# B&R Automation Studio project MappAssetInt (part 2)

#### exAssetIntCore.st
```iecst
// -------------------------------------------------------------------------------------------
// Core function block
FUNCTION_BLOCK exAssetIntCore
	// -------------------------------------------------------------------------------------------
	// Reset everything when enable is false
	IF NOT Enable THEN
		Active := FALSE;
		exLink.IsCoreActive := FALSE;
		StatusID := ERR_FUB_ENABLE_FALSE;
		Internal.State := exASSETINT_STATE_INIT_1;
		CreateLoggerEntry(exASSETINT_LOG_INFO, ADR('function block disabled'), Logger);
		RETURN;
	END_IF

	CASE Internal.State OF

		// -------------------------------------------------------------------------------------------
		// Wait for enable
		// -------------------------------------------------------------------------------------------
		exASSETINT_STATE_INIT_1:
			IF Enable THEN
				CreateLoggerEntry(exASSETINT_LOG_INFO, ADR('function block enabled'), Logger);

				// Make sure we have remanent buffer
				IF ADR(exLink) = 0 THEN
					// Set status, remember state, go to error state
					StatusID := CreateErrorState(ERR_ASSET_LINK, ADR('ERR: exLink is 0'), Logger, exCOM_SEV_ERROR,  ADR(Internal.State), ADR(Info.Diag.StatusID));
					RETURN;
				END_IF
				// Make sure we have a configuration
				IF ADR(Configuration) = 0 THEN
					// Set status, remember state, go to error state
					StatusID := CreateErrorState(ERR_ASSET_LINK, ADR('ERR: No configuation attached'), Logger, exCOM_SEV_ERROR,  ADR(Internal.State), ADR(Info.Diag.StatusID));
					RETURN;
				END_IF

				// -------------------------------------------------------------------------------------------
				// Transfer start values
				exLink.RecordCount := 0;
				exLink.JobStatistics.JobName := Parameters.Job;
				exLink.JobStatistics.CurrentUser := Parameters.CurrentUser;
				exLink.JobStatistics.AdditionalData := Parameters.AdditionalData;
				Internal.JobPieceCounterOld := PieceCounter;
				Internal.JobRejectCounterOld := RejectCounter;

				exLink.ShiftStatistics.CurrentUser := Parameters.CurrentUser;
				exLink.ShiftStatistics.AdditionalData := Parameters.AdditionalData;
				Internal.ShiftPieceCounterOld := PieceCounter;
				Internal.ShiftRejectCounterOld := RejectCounter;

				// -------------------------------------------------------------------------------------------
				// Reset error, status and function and internal blocks
				Error := FALSE;
				StatusID := ERR_OK;
				Internal.CreateDirStructure(Enable := FALSE);
				Internal.CreateMemory(Enable := FALSE);
				Internal.ReadEventData(Enable := FALSE);
				Internal.WriteEventData(Enable := FALSE);
				Internal.ReadEventData(Enable := FALSE);
				Internal.WriteEventData(Enable := FALSE);

				// -------------------------------------------------------------------------------------------
				// Check shift configuration for errors
				IF NOT exAssetIntCheckShiftData(Configuration, Logger, ADR(Internal.State), ADR(StatusID), ADR(Info.Diag.StatusID)) THEN
					RETURN;
				END_IF

				// -------------------------------------------------------------------------------------------
				// Create folder structure and read event data only after boot
				IF Internal.InitAfterBoot THEN
					Internal.State := exASSETINT_STATE_INIT_4;
				ELSE
					Internal.State := exASSETINT_STATE_INIT_2;
				END_IF
			END_IF

			// -------------------------------------------------------------------------------------------
			// Create folder structure
			// -------------------------------------------------------------------------------------------
		exASSETINT_STATE_INIT_2:
			Internal.CreateDirStructure.Enable := TRUE;
			Internal.CreateDirStructure.Device := DeviceName;
			Internal.CreateDirStructure.Logger := Logger;
			Internal.CreateDirStructure();

			// -------------------------------------------------------------------------------------------
			// Folder structure successful created
			IF Internal.CreateDirStructure.Status = ERR_OK THEN
				CreateLoggerEntry(exASSETINT_LOG_INFO, ADR('create folder structure ok'), Logger);
				Internal.State := exASSETINT_STATE_INIT_3;

				// Error
			ELSIF Internal.CreateDirStructure.Status <> ERR_FUB_BUSY THEN
				// Set status, remember state, go to error state
				StatusID := CreateErrorState(Internal.CreateDirStructure.Status, ADR('ERR: create folder structure'), Logger, exCOM_SEV_ERROR,  ADR(Internal.State), ADR(Info.Diag.StatusID));
			END_IF

			// -------------------------------------------------------------------------------------------
			// Create internal memory
			// -------------------------------------------------------------------------------------------
		exASSETINT_STATE_INIT_3:
			Internal.CreateMemory.Enable := TRUE;
			Internal.CreateMemory.Size := CORE_EVENT_NUM_MAX*SIZEOF(Internal.RecordData);
			Internal.CreateMemory.Logger := Logger;
			Internal.CreateMemory();

			// -------------------------------------------------------------------------------------------
			// Memory structure successful created
			IF Internal.CreateMemory.Status = ERR_OK THEN
				CreateLoggerEntry(exASSETINT_LOG_INFO, ADR('create internal memory ok'), Logger);
				exLink.MemoryDb := Internal.CreateMemory.MemoryDb;
				exLink.MemoryJob := Internal.CreateMemory.MemoryJob;
				exLink.MemoryShift := Internal.CreateMemory.MemoryShift;
				exLink.MemoryTimeline := Internal.CreateMemory.MemoryTimeline;
				Internal.InitAfterBoot := TRUE;
				Internal.State := exASSETINT_STATE_INIT_4;

				// Error
			ELSIF Internal.CreateMemory.Status <> ERR_FUB_BUSY THEN
				// Set status, remember state, go to error state
				StatusID := CreateErrorState(Internal.CreateMemory.Status, ADR('ERR: create internal memory'), Logger, exCOM_SEV_ERROR,  ADR(Internal.State), ADR(Info.Diag.StatusID));
			END_IF

			// -------------------------------------------------------------------------------------------
			// Read event data
			// -------------------------------------------------------------------------------------------
		exASSETINT_STATE_INIT_4:
			Internal.ReadEventData.Enable := TRUE;
			Internal.ReadEventData.Device := DeviceName;
			Internal.ReadEventData.Memory := exLink.MemoryDb;
			Internal.ReadEventData.Logger := Logger;
			Internal.ReadEventData();

			// Read events successful
			IF Internal.ReadEventData.Status = ERR_OK THEN
				CreateLoggerEntry(exASSETINT_LOG_INFO, ADR('read stored events ok'), Logger);

				// -------------------------------------------------------------------------------------------
				// Get record count, calculate next entry
				exLink.RecordCount := Internal.ReadEventData.RecordCount;
				IF exLink.RecordCount > 0 THEN
					// Get last entry, make correction if necessary
					brsmemcpy(ADR(Internal.RecordData), exLink.MemoryDb + (exLink.RecordCount - 1)*SIZEOF(Internal.RecordData), SIZEOF(Internal.RecordData));
					brsstrcpy(ADR(Internal.TmpStr1), ADR(Internal.RecordData.FileName) + FindInstr(ADR(Internal.RecordData.FileName), ADR('#')) + 1);
					Internal.RecordNext := DINT_TO_UINT(brsatoi(ADR(Internal.TmpStr1))) + 1;
					IF Internal.RecordNext >= CORE_EVENT_NUM_MAX THEN
						Internal.RecordNext := 0;
					END_IF
				END_IF

				// -------------------------------------------------------------------------------------------
				// Remember start called time
				Internal.TimeLastCallShift := clock_ms();
				Internal.TimeLastCallProduction := clock_ms();

				// -------------------------------------------------------------------------------------------
				// Refresh UI data, finish up
				exLink.RefreshJobUI := TRUE;
				exLink.RefreshShiftUI := TRUE;
				exLink.RefreshTimelineUI := TRUE;
				Internal.State := exASSETINT_STATE_IDLE;

				// Error
			ELSIF Internal.ReadEventData.Status <> ERR_FUB_BUSY THEN
				// Set status, remember state, go to error state
				StatusID := CreateErrorState(Internal.ReadEventData.Status, ADR('ERR: read stored events'), Logger, exCOM_SEV_ERROR,  ADR(Internal.State), ADR(Info.Diag.StatusID));
			END_IF

			// -------------------------------------------------------------------------------------------
			// Wait for new event
			// -------------------------------------------------------------------------------------------
		exASSETINT_STATE_IDLE:
			// Set core active, reset read write function blocks
			Active := TRUE;
			exLink.IsCoreActive := TRUE;
			Internal.ReadEventData(Enable := FALSE);
			Internal.WriteEventData(Enable := FALSE);

			// Update time information
			Internal.DTGetTime_0(enable := TRUE);
			DT_TO_DTStructure(Internal.DTGetTime_0.DT1, ADR(Internal.DT_TO_DTStructure_0));
			Internal.TimeOfDay := UDINT_TO_TOD((USINT_TO_UDINT(Internal.DT_TO_DTStructure_0.hour) * 3600000) + (USINT_TO_UDINT(Internal.DT_TO_DTStructure_0.minute) * 60000) + (USINT_TO_UDINT(Internal.DT_TO_DTStructure_0.second) * 1000));

			// Set stats timer
			Internal.StatsRefresh.IN := TRUE;
			Internal.StatsRefresh.PT := Configuration.CalculationTimeBase/10;
			Internal.StatsRefresh();

			// -------------------------------------------------------------------------------------------
			// Track current shift
			Internal.ShiftName := '';
			Internal.ShiftId := -1;
			FOR Internal.x := 0 TO SIZEOF(Configuration.Shifts)/SIZEOF(Configuration.Shifts[0]) - 1 DO
				// Shift ends on same day
				IF Configuration.Shifts[Internal.x].TotalTime.Start < Configuration.Shifts[Internal.x].TotalTime.End THEN
					IF Internal.TimeOfDay >= Configuration.Shifts[Internal.x].TotalTime.Start AND Internal.TimeOfDay <= Configuration.Shifts[Internal.x].TotalTime.End THEN
						Internal.ShiftName := Configuration.Shifts[Internal.x].Name;
						Internal.ShiftId := UINT_TO_SINT(Internal.x);
						EXIT;
					END_IF
					// Shift ends next day
				ELSE
					IF Internal.TimeOfDay >= Configuration.Shifts[Internal.x].TotalTime.Start OR Internal.TimeOfDay <= Configuration.Shifts[Internal.x].TotalTime.End THEN
						Internal.ShiftName := Configuration.Shifts[Internal.x].Name;
						Internal.ShiftId := UINT_TO_SINT(Internal.x);
						EXIT;
					END_IF
				END_IF
			END_FOR;

			// -------------------------------------------------------------------------------------------
			// Track current shift scheduled downtime
			IF exLink.ShiftId >= 0 THEN
				FOR Internal.x := 0 TO SIZEOF(Configuration.Shifts[exLink.ShiftId].ScheduledDowntime)/SIZEOF(Configuration.Shifts[exLink.ShiftId].ScheduledDowntime[0]) - 1 DO
					// Make sure we have a valid configuration
					IF TOD_TO_UDINT(Configuration.Shifts[exLink.ShiftId].ScheduledDowntime[Internal.x].Start) <> 0 OR TOD_TO_UDINT(Configuration.Shifts[exLink.ShiftId].ScheduledDowntime[Internal.x].End) <> 0 THEN
						// Downtime ends on same day
						IF Configuration.Shifts[exLink.ShiftId].ScheduledDowntime[Internal.x].Start < Configuration.Shifts[exLink.ShiftId].ScheduledDowntime[Internal.x].End THEN
							IF Internal.TimeOfDay >= Configuration.Shifts[exLink.ShiftId].ScheduledDowntime[Internal.x].Start AND Internal.TimeOfDay < Configuration.Shifts[exLink.ShiftId].ScheduledDowntime[Internal.x].End THEN
								Downtime := exASSETINT_SCHEDULED_DOWNTIME;
								DowntimeReason := Configuration.Shifts[exLink.ShiftId].ScheduledDowntime[Internal.x].Reason;
								EXIT;
							END_IF
						ELSE
							IF Internal.TimeOfDay >= Configuration.Shifts[exLink.ShiftId].ScheduledDowntime[Internal.x].Start OR Internal.TimeOfDay < Configuration.Shifts[exLink.ShiftId].ScheduledDowntime[Internal.x].End THEN
								Downtime := exASSETINT_SCHEDULED_DOWNTIME;
								DowntimeReason := Configuration.Shifts[exLink.ShiftId].ScheduledDowntime[Internal.x].Reason;
								EXIT;
							END_IF
						END_IF
					END_IF
				END_FOR;
			END_IF

			// -------------------------------------------------------------------------------------------
			// Handle shift change
			IF exLink.ShiftStatistics.ShiftName <> Internal.ShiftName THEN
				// Transfer stats to record, make sure structures are allignent
				brsmemset(ADR(Internal.RecordData), 0, SIZEOF(Internal.RecordData));

				IF Internal.ShiftName <> '' THEN
					Internal.TmpStr1 := 'new shift started ';
					brsstrcat(ADR(Internal.TmpStr1), ADR(Internal.ShiftName));
					CreateLoggerEntry(exASSETINT_LOG_INFO, ADR(Internal.TmpStr1), Logger);
				ELSIF exLink.ShiftStatistics.ShiftName <> '' THEN
					Internal.TmpStr1 := 'shift ended ';
					brsstrcat(ADR(Internal.TmpStr1), ADR(exLink.ShiftStatistics.ShiftName));
					CreateLoggerEntry(exASSETINT_LOG_INFO, ADR(Internal.TmpStr1), Logger);
				END_IF

				// Only store data when shift name was not empty
				IF exLink.ShiftStatistics.ShiftName <> '' THEN
					// Collect data for record
					Internal.RecordData.EventType := RecordTypeShift;
					Internal.RecordData.TimeStart := exLink.ShiftStatistics.StartTime;
					Internal.DT_TO_DTStructure_0.hour := UDINT_TO_USINT(TOD_TO_UDINT(Configuration.Shifts[exLink.ShiftId].TotalTime.End)/3600000);
					Internal.DT_TO_DTStructure_0.minute := UDINT_TO_USINT((TOD_TO_UDINT(Configuration.Shifts[exLink.ShiftId].TotalTime.End) - Internal.DT_TO_DTStructure_0.hour*3600000)/60000);
					Internal.RecordData.TimeEnd := DTStructure_TO_DT(ADR(Internal.DT_TO_DTStructure_0));
					Internal.RecordData.CurrentUser := exLink.ShiftStatistics.CurrentUser;
					Internal.RecordData.AdditionalData := exLink.ShiftStatistics.AdditionalData;
					Internal.RecordData.ShiftName := exLink.ShiftStatistics.ShiftName;
					Internal.RecordData.JobName := exLink.JobStatistics.JobName;
					Internal.RecordData.TotalPieces := exLink.ShiftStatistics.TotalPieces;
					Internal.RecordData.GoodPieces := exLink.ShiftStatistics.GoodPieces;
					Internal.RecordData.RejectPieces := exLink.ShiftStatistics.RejectPieces;
					Internal.RecordData.BadPieceRate := exLink.ShiftStatistics.BadPieceRate;
					Internal.RecordData.TargetPieces := exLink.ShiftStatistics.TargetPieces;
					Internal.RecordData.TotalTime := exLink.ShiftStatistics.TotalTime;
					Internal.RecordData.ScheduledDowntime := exLink.ShiftStatistics.ScheduledDowntime;
					Internal.RecordData.UnscheduledDowntime := exLink.ShiftStatistics.UnscheduledDowntime;
					Internal.RecordData.Uptime := exLink.ShiftStatistics.Uptime;
					Internal.RecordData.GoodProductionTime := exLink.ShiftStatistics.GoodProductionTime;
					Internal.RecordData.NominalProductionTime := exLink.ShiftStatistics.NominalProductionTime;
					Internal.RecordData.NominalProductionTimeRate := exLink.ShiftStatistics.NominalProductionTimeRate;
					Internal.RecordData.UnscheduledDowntimeRate := exLink.ShiftStatistics.UnscheduledDowntimeRate;
					Internal.RecordData.CurrentProductionRate := exLink.ShiftStatistics.CurrentProductionRate;

					Internal.State := exASSETINT_STATE_STORE_EVENT;
				END_IF

				// Remember job start time
				IF exLink.JobStatistics.StartTime = DT#1970-01-01-00:00:00 THEN
					exLink.JobStatistics.StartTime := Internal.DTGetTime_0.DT1;
				END_IF

				// Reset stats
				brsmemset(ADR(Info.ShiftStatistics), 0, SIZEOF(Info.ShiftStatistics));
				brsmemset(ADR(exLink.ShiftStatistics), 0, SIZEOF(exLink.ShiftStatistics));

				exLink.ShiftTotalTime := 0;
				exLink.ShiftDowntimeScheduled := 0;
				exLink.ShiftDowntimeUnscheduled := 0;

				// Transfer data to shift stats
				exLink.ShiftId := Internal.ShiftId;
				exLink.ShiftStatistics.StartTime := Internal.DTGetTime_0.DT1;
				exLink.ShiftStatistics.ShiftName := Internal.ShiftName;
				exLink.ShiftStatistics.CurrentUser := Parameters.CurrentUser;
				exLink.ShiftStatistics.AdditionalData := Parameters.AdditionalData;
			END_IF

			// -------------------------------------------------------------------------------------------
			// Calculate shift and job statistics
			IF Internal.ShiftName <> '' THEN

				// Calculate new stats
				IF Internal.StatsRefresh.Q THEN
					// Get time difference between calls
					Internal.DiffLastCallShift := DiffT(clock_ms(), Internal.TimeLastCallShift);
					Internal.TimeLastCallShift := clock_ms();

					// Handle diff timer overflow
					IF Internal.DiffLastCallShift = 16#FFFFFFFF THEN
						CreateLoggerEntry(exASSETINT_LOG_INFO, ADR('diff timer overflow'), Logger);
					ELSE

						// Do not count when downtime is active
						IF Downtime = exASSETINT_NO_DOWNTIME THEN
							// Transfer job counter data
							IF Internal.JobPieceCounterOld <= PieceCounter THEN
								exLink.JobStatistics.TotalPieces := exLink.JobStatistics.TotalPieces + (PieceCounter - Internal.JobPieceCounterOld);
							ELSE
								CreateLoggerEntry(exASSETINT_LOG_ERROR, ADR('job piece count overflow'), Logger);
								exLink.JobStatistics.TotalPieces := exLink.JobStatistics.TotalPieces + (16#FFFFFFFF - Internal.JobPieceCounterOld + PieceCounter);
							END_IF

							IF Internal.JobRejectCounterOld <= RejectCounter THEN
								exLink.JobStatistics.RejectPieces := exLink.JobStatistics.RejectPieces + (RejectCounter - Internal.JobRejectCounterOld);
							ELSE
								CreateLoggerEntry(exASSETINT_LOG_ERROR, ADR('job reject count overflow'), Logger);
								exLink.JobStatistics.RejectPieces := exLink.JobStatistics.RejectPieces + (16#FFFFFFFF - Internal.JobRejectCounterOld + RejectCounter);
							END_IF
						END_IF
						Internal.JobPieceCounterOld := PieceCounter;
						Internal.JobRejectCounterOld := RejectCounter;
						CalcStatsJob(exLink, Internal.DiffLastCallShift, Downtime, Parameters, ADR(Info.JobStatistics));

						// Do not count when downtime is active
						IF Downtime = exASSETINT_NO_DOWNTIME THEN
							// Transfer shift counter data
							IF Internal.ShiftPieceCounterOld <= PieceCounter THEN
								exLink.ShiftStatistics.TotalPieces := exLink.ShiftStatistics.TotalPieces + (PieceCounter - Internal.ShiftPieceCounterOld);
							ELSE
								CreateLoggerEntry(exASSETINT_LOG_ERROR, ADR('shift piece count overflow'), Logger);
								exLink.ShiftStatistics.TotalPieces := exLink.ShiftStatistics.TotalPieces + (16#FFFFFFFF - Internal.ShiftPieceCounterOld + PieceCounter);
							END_IF

							IF Internal.ShiftRejectCounterOld <= RejectCounter THEN
								exLink.ShiftStatistics.RejectPieces := exLink.ShiftStatistics.RejectPieces + (RejectCounter - Internal.ShiftRejectCounterOld);
							ELSE
								CreateLoggerEntry(exASSETINT_LOG_ERROR, ADR('shift reject count overflow'), Logger);
								exLink.ShiftStatistics.RejectPieces := exLink.ShiftStatistics.RejectPieces + (16#FFFFFFFF - Internal.ShiftRejectCounterOld + RejectCounter);
							END_IF
						END_IF
						Internal.ShiftPieceCounterOld := PieceCounter;
						Internal.ShiftRejectCounterOld := RejectCounter;
						CalcStatsShift(exLink, Internal.DiffLastCallShift, Downtime, Parameters, ADR(Info.ShiftStatistics));

						// Transfer shift data to main function block
						CurrentProductionRate := exLink.ShiftStatistics.CurrentProductionRate;
						NominalProductionTimeRate := exLink.ShiftStatistics.NominalProductionTimeRate;
						BadPieceRate := exLink.ShiftStatistics.BadPieceRate;
						ScheduledDowntimeRate := exLink.ShiftStatistics.ScheduledDowntimeRate;
						UnscheduledDowntimeRate := exLink.ShiftStatistics.UnscheduledDowntimeRate;

					END_IF
				END_IF

				// When no shift is active
			ELSE
				// Dont count when no shift is active, reset last call
				Internal.ShiftPieceCounterOld := PieceCounter;
				Internal.ShiftRejectCounterOld := RejectCounter;
				Internal.JobPieceCounterOld := PieceCounter;
				Internal.JobRejectCounterOld := RejectCounter;

				Internal.TimeLastCallShift := clock_ms();
			END_IF

			// -------------------------------------------------------------------------------------------
			// Handle production state change
			IF Internal.State <> exASSETINT_STATE_STORE_EVENT THEN
				IF (exLink.ShiftStatistics.ShiftName <> exLink.ProductionShiftName) OR (exLink.JobStatistics.JobName <> exLink.ProductionJobName AND exLink.ShiftId >= 0) OR (Downtime <> exLink.ProductionDowntime AND exLink.ShiftId >= 0) THEN
					// Create log message
					Internal.TmpStr1 := 'production state changed from ';
					IF exLink.ProductionState = exASSETINT_STATE_NO_SHIFT_ACTIVE THEN
						brsstrcat(ADR(Internal.TmpStr1), ADR('no shift to '));
					ELSIF exLink.ProductionState = exASSETINT_STATE_UPTIME THEN
						brsstrcat(ADR(Internal.TmpStr1), ADR('uptime to '));
					ELSIF exLink.ProductionState = exASSETINT_STATE_SCHDL_DOWNTIME THEN
						brsstrcat(ADR(Internal.TmpStr1), ADR('scheduled dt to '));
					ELSE
						brsstrcat(ADR(Internal.TmpStr1), ADR('unscheduled dt to '));
					END_IF

					// Transfer stats to record, make sure structures are allignent
					brsmemset(ADR(Internal.RecordData), 0, SIZEOF(Internal.RecordData));

					// Collect data for record
					Internal.RecordData.TimeStart := exLink.ProductionStateStart;
					Internal.RecordData.TimeEnd := Internal.DTGetTime_0.DT1;
					Internal.RecordData.ShiftName := exLink.ProductionShiftName;
					Internal.RecordData.JobName := exLink.ProductionJobName;
					Internal.RecordData.EventType := UDINT_TO_UINT(exLink.ProductionState + 2);

					Internal.ProductionTotalTime := LREAL_TO_UDINT(exLink.ProductionTotalTime/1000);
					Internal.RecordData.TotalTime.Hours := Internal.ProductionTotalTime/3600;
					Internal.RecordData.TotalTime.Minutes := UDINT_TO_USINT((Internal.ProductionTotalTime - Internal.RecordData.TotalTime.Hours*3600)/60);
					Internal.RecordData.TotalTime.Seconds := UDINT_TO_USINT(Internal.ProductionTotalTime - Internal.RecordData.TotalTime.Hours*3600 - Internal.RecordData.TotalTime.Minutes*60);

					// State change is new job
					IF (exLink.JobStatistics.JobName <> exLink.ProductionJobName) THEN
						brsstrcat(ADR(Internal.TmpStr1), ADR('new job > '));
						brsstrcat(ADR(Internal.TmpStr1), ADR(exLink.JobStatistics.JobName));
						exLink.ProductionState := exASSETINT_STATE_UPTIME;

						// State change is to no shift
					ELSIF (exLink.ProductionShiftName <> '' AND exLink.ShiftStatistics.ShiftName = '') THEN
						brsstrcat(ADR(Internal.TmpStr1), ADR('no shift'));
						exLink.ProductionState := exASSETINT_STATE_NO_SHIFT_ACTIVE;

						// State change is to uptime
					ELSIF (exLink.ProductionShiftName = '' AND exLink.ShiftStatistics.ShiftName <> '') THEN
						brsstrcat(ADR(Internal.TmpStr1), ADR('uptime'));
						exLink.ProductionState := exASSETINT_STATE_UPTIME;

						// State is shift change
					ELSIF (exLink.ProductionShiftName <> exLink.ShiftStatistics.ShiftName) THEN
						brsstrcat(ADR(Internal.TmpStr1), ADR('new shift'));
						exLink.ProductionState := exASSETINT_STATE_UPTIME;

						// State change is downtime
					ELSE
						IF Downtime = exASSETINT_NO_DOWNTIME THEN
							brsstrcat(ADR(Internal.TmpStr1), ADR('no downtime'));
						ELSIF Downtime = exASSETINT_SCHEDULED_DOWNTIME THEN
							brsstrcat(ADR(Internal.TmpStr1), ADR('scheduled dt > '));
							brsstrcat(ADR(Internal.TmpStr1), ADR(DowntimeReason));
						ELSE
							brsstrcat(ADR(Internal.TmpStr1), ADR('unscheduled dt > '));
							brsstrcat(ADR(Internal.TmpStr1), ADR(DowntimeReason));
						END_IF

						IF exLink.ProductionState = exASSETINT_STATE_SCHDL_DOWNTIME OR exLink.ProductionState = exASSETINT_STATE_UNSCH_DOWNTIME THEN
							Internal.RecordData.AdditionalData := DowntimeReason;
						END_IF
						exLink.ProductionState := UDINT_TO_UINT(Downtime + 1);
					END_IF
					CreateLoggerEntry(exASSETINT_LOG_INFO, ADR(Internal.TmpStr1), Logger);

					exLink.ProductionShiftName :=exLink.ShiftStatistics.ShiftName;
					exLink.ProductionJobName := exLink.JobStatistics.JobName;
					exLink.ProductionDowntime := Downtime;

					// Skip after cold start
					IF exLink.ProductionStateStart <> DT#1970-01-01-00:00:00 THEN
						exLink.ProductionStateStart := Internal.DTGetTime_0.DT1;
						exLink.ProductionTotalTime := 0;

						// Create new event
						Internal.State := exASSETINT_STATE_STORE_EVENT;

						// Just remember start time after cold start
					ELSE
						exLink.ProductionStateStart := Internal.DTGetTime_0.DT1;
					END_IF

				END_IF
			END_IF
			// Remember production duration
			IF Internal.StatsRefresh.Q THEN
				// Get time difference between calls
				Internal.DiffLastCallProduction := DiffT(clock_ms(), Internal.TimeLastCallProduction);
				Internal.TimeLastCallProduction := clock_ms();
				IF Internal.DiffLastCallProduction = 16#FFFFFFFF THEN
					CreateLoggerEntry(exASSETINT_LOG_INFO, ADR('diff timer overflow'), Logger);
				ELSE
					exLink.ProductionTotalTime := exLink.ProductionTotalTime + Internal.DiffLastCallProduction;
				END_IF
			END_IF

			// -------------------------------------------------------------------------------------------
			// Handle update command
			IF EDGEPOS(Update) THEN
				CreateLoggerEntry(exASSETINT_LOG_INFO, ADR('update command triggered'), Logger);

				// -------------------------------------------------------------------------------------------
				// Check shift configuration for errors
				IF NOT exAssetIntCheckShiftData(Configuration, Logger, ADR(Internal.State), ADR(StatusID), ADR(Info.Diag.StatusID)) THEN
					RETURN;
				END_IF

				// Job has changed
				IF Parameters.Job <> exLink.JobStatistics.JobName THEN
					Internal.TmpStr1 := 'new job started ';
					brsstrcat(ADR(Internal.TmpStr1), ADR(Parameters.Job));
					CreateLoggerEntry(exASSETINT_LOG_INFO, ADR(Internal.TmpStr1), Logger);

					CommandBusy := TRUE;
					CommandDone := FALSE;
					UpdateDone := FALSE;

					// Transfer stats to record, make sure structures are allignent
					brsmemset(ADR(Internal.RecordData), 0, SIZEOF(Internal.RecordData));

					// Collect data for record
					Internal.RecordData.EventType := RecordTypeJob;
					Internal.RecordData.TimeStart := exLink.JobStatistics.StartTime;
					Internal.RecordData.TimeEnd := Internal.DTGetTime_0.DT1;
					Internal.RecordData.CurrentUser := exLink.JobStatistics.CurrentUser;
					Internal.RecordData.AdditionalData := exLink.JobStatistics.AdditionalData;
					Internal.RecordData.ShiftName := exLink.ShiftStatistics.ShiftName;
					Internal.RecordData.JobName := exLink.JobStatistics.JobName;
					Internal.RecordData.TotalPieces := exLink.JobStatistics.TotalPieces;
					Internal.RecordData.GoodPieces := exLink.JobStatistics.GoodPieces;
					Internal.RecordData.RejectPieces := exLink.JobStatistics.RejectPieces;
					Internal.RecordData.BadPieceRate := exLink.JobStatistics.BadPieceRate;
					Internal.RecordData.TotalTime := exLink.JobStatistics.TotalTime;
					Internal.RecordData.ScheduledDowntime := exLink.JobStatistics.ScheduledDowntime;
					Internal.RecordData.UnscheduledDowntime := exLink.JobStatistics.UnscheduledDowntime;
					Internal.RecordData.Uptime := exLink.JobStatistics.Uptime;
					Internal.RecordData.GoodProductionTime := exLink.JobStatistics.GoodProductionTime;
					Internal.RecordData.NominalProductionTime := exLink.JobStatistics.NominalProductionTime;
					Internal.RecordData.NominalProductionTimeRate := exLink.JobStatistics.NominalProductionTimeRate;
					Internal.RecordData.UnscheduledDowntimeRate := exLink.JobStatistics.UnscheduledDowntimeRate;
					Internal.RecordData.CurrentProductionRate := exLink.JobStatistics.CurrentProductionRate;

					// Reset stats and remember new start time
					brsmemset(ADR(Info.JobStatistics), 0, SIZEOF(Info.JobStatistics));
					brsmemset(ADR(exLink.JobStatistics), 0, SIZEOF(exLink.JobStatistics));

					exLink.JobTotalTime := 0;
					exLink.JobDowntimeScheduled := 0;
					exLink.JobDowntimeUnscheduled := 0;

					// Transfer data to job stats
					exLink.JobStatistics.StartTime := Internal.DTGetTime_0.DT1;
					exLink.JobStatistics.JobName := Parameters.Job;
					exLink.JobStatistics.CurrentUser := Parameters.CurrentUser;
					exLink.JobStatistics.AdditionalData := Parameters.AdditionalData;

					Internal.State := exASSETINT_STATE_STORE_EVENT;
				ELSE
					CommandBusy := FALSE;
					CommandDone := TRUE;
					UpdateDone := TRUE;
				END_IF
			END_IF

			IF NOT Update THEN
				UpdateDone := FALSE;
			END_IF

			// -------------------------------------------------------------------------------------------
			// Handle reset command
			IF EDGEPOS(Reset) THEN
				CreateLoggerEntry(exASSETINT_LOG_INFO, ADR('reset command triggered'), Logger);

				CommandBusy := TRUE;
				CommandDone := FALSE;

				// Reset stats
				brsmemset(ADR(Info.JobStatistics), 0, SIZEOF(Info.JobStatistics));
				brsmemset(ADR(exLink.JobStatistics), 0, SIZEOF(exLink.JobStatistics));

				exLink.JobTotalTime := 0;
				exLink.JobDowntimeScheduled := 0;
				exLink.JobDowntimeUnscheduled := 0;

				// Transfer data to job stats
				exLink.JobStatistics.StartTime := Internal.DTGetTime_0.DT1;
				exLink.JobStatistics.JobName := Parameters.Job;
				exLink.JobStatistics.CurrentUser := Parameters.CurrentUser;
				exLink.JobStatistics.AdditionalData := Parameters.AdditionalData;

				// Reset stats
				brsmemset(ADR(Info.ShiftStatistics), 0, SIZEOF(Info.ShiftStatistics));
				brsmemset(ADR(exLink.ShiftStatistics), 0, SIZEOF(exLink.ShiftStatistics));

				exLink.ShiftTotalTime := 0;
				exLink.ShiftDowntimeScheduled := 0;
				exLink.ShiftDowntimeUnscheduled := 0;

				// Transfer data to shift stats
				exLink.ShiftId := Internal.ShiftId;
				exLink.ShiftStatistics.StartTime := Internal.DTGetTime_0.DT1;
				exLink.ShiftStatistics.ShiftName := Internal.ShiftName;
				exLink.ShiftStatistics.CurrentUser := Parameters.CurrentUser;
				exLink.ShiftStatistics.AdditionalData := Parameters.AdditionalData;

				CommandBusy := FALSE;
				CommandDone := TRUE;
			END_IF

			// -------------------------------------------------------------------------------------------
			// Handle export command
			IF EDGEPOS(Export) THEN

				CommandBusy := TRUE;
				CommandDone := FALSE;
				ExportDone := FALSE;

				Internal.State := exASSETINT_STATE_EXPORT_EVENTS;
			END_IF

			IF NOT Export THEN
				ExportDone := FALSE;
			END_IF

			// -------------------------------------------------------------------------------------------
			// Reset refresh timer
			IF Internal.StatsRefresh.Q THEN
				// Set stats timer
				Internal.StatsRefresh.IN := FALSE;
				Internal.StatsRefresh();
			END_IF

			IF Update = FALSE AND Export = FALSE AND Reset = FALSE THEN
				CommandDone := FALSE;
			END_IF

			// -------------------------------------------------------------------------------------------
			// Store new event
			// -------------------------------------------------------------------------------------------
		exASSETINT_STATE_STORE_EVENT:
			Internal.WriteEventData.Enable := TRUE;
			Internal.WriteEventData.Device := StorageName;
			Internal.WriteEventData.Logger := Logger;
			Internal.WriteEventData.RecordData := ADR(Internal.RecordData);
			Internal.WriteEventData.RecordNext := Internal.RecordNext;
			Internal.WriteEventData();

			// -------------------------------------------------------------------------------------------
			// Event successful created
			IF Internal.WriteEventData.Status = ERR_OK THEN
				CreateLoggerEntry(exASSETINT_LOG_INFO, ADR('create new event ok'), Logger);

				// Calculate new last record and record count
				Internal.RecordNext := Internal.RecordNext + 1;
				IF Internal.RecordNext >= CORE_EVENT_NUM_MAX THEN
					Internal.RecordNext := 0;
				END_IF
				// Copy new record into memeory
				IF exLink.RecordCount < CORE_EVENT_NUM_MAX THEN
					exLink.RecordCount := exLink.RecordCount + 1;
				ELSE
					brsmemmove(exLink.MemoryDb, exLink.MemoryDb + SIZEOF(Internal.RecordData), SIZEOF(Internal.RecordData)*(exLink.RecordCount - 1));
				END_IF
				brsmemcpy(exLink.MemoryDb + SIZEOF(Internal.RecordData)*(exLink.RecordCount - 1), ADR(Internal.RecordData), SIZEOF(Internal.RecordData));

				// Refrehs UI data, finish up
				exLink.RefreshJobUI := TRUE;
				exLink.RefreshShiftUI := TRUE;
				exLink.RefreshTimelineUI := TRUE;

				UpdateDone := TRUE;
				CommandBusy := FALSE;
				CommandDone := TRUE;

				StatusID := ERR_OK;
				Internal.State := exASSETINT_STATE_IDLE;

				// Error
			ELSIF Internal.WriteEventData.Status <> ERR_FUB_BUSY THEN
				// Set status, remember state, go to error state
				StatusID := CreateErrorState(Internal.WriteEventData.Status, ADR('ERR: create new event'), Logger, exCOM_SEV_ERROR,  ADR(Internal.State), ADR(Info.Diag.StatusID));
			END_IF

			// -------------------------------------------------------------------------------------------
			// Export all events
			// -------------------------------------------------------------------------------------------
		exASSETINT_STATE_EXPORT_EVENTS:
			Internal.ExportEventData.Enable := TRUE;
			Internal.ExportEventData.Device := DeviceName;
			Internal.ExportEventData.Logger := Logger;
			Internal.ExportEventData.RecordCount := exLink.RecordCount;
			Internal.ExportEventData.Memory := exLink.MemoryDb;
			Internal.ExportEventData.Configuration := Configuration.Export;
			Internal.ExportEventData();

			// -------------------------------------------------------------------------------------------
			// Event successful created
			IF Internal.ExportEventData.Status = ERR_OK THEN
				CreateLoggerEntry(exASSETINT_LOG_INFO, ADR('export events ok'), Logger);

				ExportDone := TRUE;
				CommandBusy := FALSE;
				CommandDone := TRUE;

				StatusID := ERR_OK;
				Internal.State := exASSETINT_STATE_IDLE;

				// Error
			ELSIF Internal.ExportEventData.Status <> ERR_FUB_BUSY THEN
				// Set status, remember state, go to error state
				StatusID := CreateErrorState(Internal.ExportEventData.Status, ADR('ERR: export events'), Logger, exCOM_SEV_ERROR,  ADR(Internal.State), ADR(Info.Diag.StatusID));
			END_IF

			// -------------------------------------------------------------------------------------------
			// Error state
			// -------------------------------------------------------------------------------------------
		exASSETINT_STATE_ERROR:

			// Reset error state
			IF EDGEPOS(ErrorReset) THEN
				Internal.StateError := exASSETINT_STATE_NONE;
				Internal.State := exASSETINT_STATE_INIT_1;
			END_IF
	END_CASE;

END_FUNCTION_BLOCK
```

#### exAssetIntCoreConfig.st
```iecst
// -------------------------------------------------------------------------------------------
// File version 1004
// -------------------------------------------------------------------------------------------
// Config function block
FUNCTION_BLOCK exAssetIntCoreConfig
	// -------------------------------------------------------------------------------------------
	// Reset everything when enable is false
	IF NOT Enable THEN
		Active := FALSE;
		StatusID := ERR_FUB_ENABLE_FALSE;
		Internal.State := exASSETINT_STATE_INIT_1;
		CreateLoggerEntry(exASSETINT_LOG_INFO, ADR('function block disabled'), Logger);
		RETURN;
	END_IF

	// -------------------------------------------------------------------------------------------
	// Permanent watch critical values
	IF Internal.State <> exASSETINT_STATE_ERROR THEN
		// Make sure we have a configuration
		IF ADR(Configuration) = 0 THEN
			// Set status, remember state, go to error state
			StatusID := CreateErrorState(ERR_ASSET_LINK, ADR('ERR: No configuation attached'), Logger, exCOM_SEV_ERROR, ADR(Internal.State), ADR(Info.Diag.StatusID));
			RETURN;
		END_IF
		// Make sure we have a device name
		IF ADR(DeviceName) = 0 THEN
			// Set status, remember state, go to error state
			StatusID := CreateErrorState(ERR_ASSET_LINK, ADR('ERR: No device name attached'), Logger, exCOM_SEV_ERROR, ADR(Internal.State), ADR(Info.Diag.StatusID));
			RETURN;
		END_IF
	END_IF

	CASE Internal.State OF

		// -------------------------------------------------------------------------------------------
		// Wait for enable
		exASSETINT_STATE_INIT_1:
			IF Enable THEN
				CreateLoggerEntry(exASSETINT_LOG_INFO, ADR('function block enabled'), Logger);

				// Reset error and status
				brsmemset(ADR(Info.Diag), 0, SIZEOF(Info.Diag));
				Error := FALSE;
				StatusID := ERR_OK;
				CommandBusy := FALSE;
				CommandDone := FALSE;

				Internal.State := exASSETINT_STATE_IDLE;
			END_IF

			// -------------------------------------------------------------------------------------------
			// Wait for new event
		exASSETINT_STATE_IDLE:
			Active := TRUE;

			// Handle configuration load command
			IF EDGEPOS(Load) THEN
				CreateLoggerEntry(exASSETINT_LOG_INFO, ADR('command load configuration'), Logger);
				CommandBusy := TRUE;
				CommandDone := FALSE;

				Internal.State := exASSETINT_STATE_LOAD_CFG;
			END_IF

			// Handle configuration save command
			IF EDGEPOS(Save) THEN
				CreateLoggerEntry(exASSETINT_LOG_INFO, ADR('command save configuration'), Logger);
				CommandBusy := TRUE;
				CommandDone := FALSE;

				Internal.State := exASSETINT_STATE_SAVE_CFG;
			END_IF

			IF Load = FALSE AND Save = FALSE THEN
				CommandDone := FALSE;
			END_IF

		// -------------------------------------------------------------------------------------------
		// Load configuration
		exASSETINT_STATE_LOAD_CFG:
			Internal.ReadConfiguration.Enable := TRUE;
			Internal.ReadConfiguration.Device := ADR(DeviceName);
			Internal.ReadConfiguration.Logger := Logger;
			Internal.ReadConfiguration();

			// Event successful created
			IF Internal.ReadConfiguration.Status = ERR_OK THEN
				CreateLoggerEntry(exASSETINT_LOG_INFO, ADR('load configuration ok'), Logger);
				Configuration := Internal.ReadConfiguration.Configuration;

				CommandBusy := FALSE;
				CommandDone := TRUE;
				StatusID := ERR_OK;

				Internal.State := exASSETINT_STATE_IDLE;

			// Error
			ELSIF Internal.ReadConfiguration.Status <> ERR_FUB_BUSY THEN
				// Set status, remember state, go to error state
				StatusID := CreateErrorState(Internal.ReadConfiguration.Status, ADR('ERR: load configuration'), Logger, exCOM_SEV_ERROR,  ADR(Internal.State), ADR(Info.Diag.StatusID));
			END_IF

			// -------------------------------------------------------------------------------------------
			// Save configuration
		exASSETINT_STATE_SAVE_CFG:
			Internal.WriteConfiguration.Enable := TRUE;
			Internal.WriteConfiguration.Device := ADR(DeviceName);
			Internal.WriteConfiguration.Logger := Logger;
			Internal.WriteConfiguration.Configuration := Configuration;
			Internal.WriteConfiguration();

			// Event successful created
			IF Internal.WriteConfiguration.Status = ERR_OK THEN
				CreateLoggerEntry(exASSETINT_LOG_INFO, ADR('save configuration ok'), Logger);

				CommandBusy := FALSE;
				CommandDone := TRUE;
				StatusID := ERR_OK;

				Internal.State := exASSETINT_STATE_IDLE;

			// Error
			ELSIF Internal.WriteConfiguration.Status <> ERR_FUB_BUSY THEN
				// Set status, remember state, go to error state
				StatusID := CreateErrorState(Internal.WriteConfiguration.Status, ADR('ERR: save configuration'), Logger, exCOM_SEV_ERROR,  ADR(Internal.State), ADR(Info.Diag.StatusID));
			END_IF

		// -------------------------------------------------------------------------------------------
		// Error state
		exASSETINT_STATE_ERROR:
			Internal.WriteConfiguration.Enable := FALSE;
			Internal.WriteConfiguration();
			Internal.ReadConfiguration.Enable := FALSE;
			Internal.ReadConfiguration();

			IF EDGEPOS(ErrorReset) THEN
				Internal.StateError := exASSETINT_STATE_NONE;
				Internal.State := exASSETINT_STATE_INIT_1;
			END_IF
	END_CASE;
END_FUNCTION_BLOCK
```

#### exAssetIntUI.st
```iecst
// -------------------------------------------------------------------------------------------
// Job UI function block
FUNCTION_BLOCK exAssetIntJobListUI
	// -------------------------------------------------------------------------------------------
	// Reset everything when enable is false
	IF NOT Enable THEN
		StatusID := ERR_FUB_ENABLE_FALSE;
		Active := FALSE;
		Internal.State := exASSETINT_STATE_INIT_1;
		CreateLoggerEntry(exASSETINT_LOG_INFO, ADR('function block disabled'), Logger);
		RETURN;
	END_IF

	CASE Internal.State OF

		// -------------------------------------------------------------------------------------------
		// Wait for enable
		exASSETINT_STATE_INIT_1:
			IF Enable THEN
				CreateLoggerEntry(exASSETINT_LOG_INFO, ADR('function block enabled'), Logger);

				// Check prerequisites, exLink and buffers
				IF NOT exAssetIntCheckPreq(exLink, Logger, ADR(Internal.State), ADR(StatusID), ADR(Info.Diag.StatusID)) THEN
					RETURN;
				END_IF

				// Reset error and status
				Error := FALSE;
				StatusID := ERR_OK;
				Internal.SortingStartTimeOld := UDINT_TO_DINT(16#FFFFFFFF);

				// Reset filter settings
				exAssetIntFilterReset(ADR(UIConnect.Filter));

				Internal.State := exASSETINT_STATE_IDLE;
			END_IF

			// -------------------------------------------------------------------------------------------
			// Wait for new event
		exASSETINT_STATE_IDLE:
			// Set status
			UIConnect.Status := exASSETINT_UI_STATUS_IDLE;
			Active := TRUE;

			// Handle dialog window
			Internal.State := exAssetIntFilterListUI(ADR(UIConnect.Filter), ADR(UIConnect.Status), Logger);

			// Handle sorting direction change
			IF UISetup.SortingStartTime <> Internal.SortingStartTimeOld AND exLink.RecordCount > 0 THEN
				Internal.State := exASSETINT_STATE_UI_BUFFER;
			END_IF
			Internal.SortingStartTimeOld := UISetup.SortingStartTime;

			// Handle page up and down
			exAssetIntScrollListUI(Internal.RecordCount, UI_JOB_LIST_IDX, ADR(UIConnect.Output.PageUp), ADR(UIConnect.Output.PageDown), ADR(UIConnect.Output.StepUp), ADR(UIConnect.Output.StepDown), ADR(Internal.RecordStart), ADR(Internal.State));

			// Wait for core task to call update command
			IF exLink.RefreshJobUI AND exLink.RecordCount > 0 THEN
				Internal.State := exASSETINT_STATE_UI_BUFFER;
			END_IF

			// -------------------------------------------------------------------------------------------
			// Copy job data from global buffer to job buffer
		exASSETINT_STATE_UI_BUFFER:
			// Set status
			CreateLoggerEntry(exASSETINT_LOG_INFO, ADR('refresh job data'), Logger);
			UIConnect.Status := exASSETINT_UI_STATUS_UPDATE;

			// Generate job data
			Internal.RecordCount := exAssetIntBufferUI(exLink.MemoryJob, exLink, UISetup.SortingStartTime, UIConnect.Filter, RecordTypeJob);

			Internal.State := exASSETINT_STATE_UI_DATA;

		// -------------------------------------------------------------------------------------------
		// Transfer data from buffer to list array
		exASSETINT_STATE_UI_DATA:

			Internal.x := 0;
			brsmemset(ADR(UIConnect.Output), 0, SIZEOF(UIConnect.Output));
			REPEAT
				brsmemcpy(ADR(Internal.RecordData), exLink.MemoryJob + (Internal.x + Internal.RecordStart)*SIZEOF(Internal.RecordData), SIZEOF(Internal.RecordData));

				UIConnect.Output.JobStartTime[Internal.x] := Internal.RecordData.TimeStart;
				UIConnect.Output.JobEndTime[Internal.x] := Internal.RecordData.TimeEnd;
				UIConnect.Output.JobName[Internal.x] := Internal.RecordData.JobName;
				UIConnect.Output.CurrentUser[Internal.x] := Internal.RecordData.CurrentUser;
				UIConnect.Output.AdditionalData[Internal.x] := Internal.RecordData.AdditionalData;
				UIConnect.Output.TotalPieces[Internal.x] := Internal.RecordData.TotalPieces;
				UIConnect.Output.GoodPieces[Internal.x] := Internal.RecordData.GoodPieces;
				UIConnect.Output.RejectPieces[Internal.x] := Internal.RecordData.RejectPieces;
				UIConnect.Output.BadPieceRate[Internal.x] := Internal.RecordData.BadPieceRate;
				UIConnect.Output.TotalTime[Internal.x] := Internal.RecordData.TotalTime;
				UIConnect.Output.ScheduledDowntime[Internal.x] := Internal.RecordData.ScheduledDowntime;
				UIConnect.Output.UnscheduledDowntime[Internal.x] := Internal.RecordData.UnscheduledDowntime;
				UIConnect.Output.Uptime[Internal.x] := Internal.RecordData.Uptime;
				UIConnect.Output.GoodProductionTime[Internal.x] := Internal.RecordData.GoodProductionTime;
				UIConnect.Output.NominalProductionTime[Internal.x] := Internal.RecordData.NominalProductionTime;
				UIConnect.Output.NominalProductionRate[Internal.x] := Internal.RecordData.NominalProductionTimeRate;
				UIConnect.Output.UnscheduledDowntimeRate[Internal.x] := Internal.RecordData.UnscheduledDowntimeRate;
				UIConnect.Output.ProductionRate[Internal.x] := Internal.RecordData.CurrentProductionRate;
				UIConnect.Output.ShiftName[Internal.x] := Internal.RecordData.ShiftName;

				Internal.x := Internal.x + 1;

				UNTIL (Internal.x = UI_JOB_LIST_IDX) OR (Internal.x + Internal.RecordStart >= Internal.RecordCount)
			END_REPEAT;

			exLink.RefreshJobUI := FALSE;
			UIConnect.Output.PageUp := FALSE;
			UIConnect.Output.PageDown := FALSE;
			UIConnect.Output.StepUp := FALSE;
			UIConnect.Output.StepDown := FALSE;

			CreateLoggerEntry(exASSETINT_LOG_INFO, ADR('refresh job done'), Logger);
			Internal.State := exASSETINT_STATE_IDLE;

		// -------------------------------------------------------------------------------------------
		// Error state
		exASSETINT_STATE_ERROR:
			IF EDGEPOS(ErrorReset) THEN
				Internal.StateError := exASSETINT_STATE_NONE;
				Internal.State := exASSETINT_STATE_INIT_1;
			END_IF
	END_CASE;
END_FUNCTION_BLOCK

// -------------------------------------------------------------------------------------------
// Shift UI function block
FUNCTION_BLOCK exAssetIntShiftListUI
	// -------------------------------------------------------------------------------------------
	// Reset everything when enable is false
	IF NOT Enable THEN
		StatusID := ERR_FUB_ENABLE_FALSE;
		Active := FALSE;
		Internal.State := exASSETINT_STATE_INIT_1;
		CreateLoggerEntry(exASSETINT_LOG_INFO, ADR('function block disabled'), Logger);
		RETURN;
	END_IF

	CASE Internal.State OF

		// -------------------------------------------------------------------------------------------
		// Wait for enable
		exASSETINT_STATE_INIT_1:
			IF Enable THEN
				CreateLoggerEntry(exASSETINT_LOG_INFO, ADR('function block enabled'), Logger);

				// Check prerequisites, exLink and buffers
				IF NOT exAssetIntCheckPreq(exLink, Logger, ADR(Internal.State), ADR(StatusID), ADR(Info.Diag.StatusID)) THEN
					RETURN;
				END_IF

				// Reset error and status
				Error := FALSE;
				StatusID := ERR_OK;
				Internal.SortingStartTimeOld := UDINT_TO_DINT(16#FFFFFFFF);

				// Reset filter settings
				exAssetIntFilterReset(ADR(UIConnect.Filter));

				Internal.State := exASSETINT_STATE_IDLE;
			END_IF

			// -------------------------------------------------------------------------------------------
			// Wait for new event
		exASSETINT_STATE_IDLE:
			// Set status
			UIConnect.Status := exASSETINT_UI_STATUS_IDLE;
			Active := TRUE;

			// Handle dialog window
			Internal.State := exAssetIntFilterListUI(ADR(UIConnect.Filter), ADR(UIConnect.Status), Logger);

			// Handle sorting direction change
			IF UISetup.SortingStartTime <> Internal.SortingStartTimeOld AND exLink.RecordCount > 0 THEN
				Internal.State := exASSETINT_STATE_UI_BUFFER;
			END_IF
			Internal.SortingStartTimeOld := UISetup.SortingStartTime;

			// Handle page up and down
			exAssetIntScrollListUI(Internal.RecordCount, UI_TIMELINE_IDX, ADR(UIConnect.Output.PageUp), ADR(UIConnect.Output.PageDown), ADR(UIConnect.Output.StepUp), ADR(UIConnect.Output.StepDown), ADR(Internal.RecordStart), ADR(Internal.State));

			// Wait for core task to call update command
			IF exLink.RefreshShiftUI AND exLink.RecordCount > 0 THEN
				Internal.State := exASSETINT_STATE_UI_BUFFER;
			END_IF

			// -------------------------------------------------------------------------------------------
			// Copy shift data from global buffer to shift buffer
		exASSETINT_STATE_UI_BUFFER:
			// Set status
			CreateLoggerEntry(exASSETINT_LOG_INFO, ADR('refresh shift data'), Logger);
			UIConnect.Status := exASSETINT_UI_STATUS_UPDATE;

			// Generate shift data
			Internal.RecordCount := exAssetIntBufferUI(exLink.MemoryShift, exLink, UISetup.SortingStartTime, UIConnect.Filter, RecordTypeShift);

			Internal.State := exASSETINT_STATE_UI_DATA;

			// -------------------------------------------------------------------------------------------
			// Transfer data from buffer to list array
		exASSETINT_STATE_UI_DATA:

			Internal.x := 0;
			brsmemset(ADR(UIConnect.Output), 0, SIZEOF(UIConnect.Output));
			REPEAT
				brsmemcpy(ADR(Internal.RecordData), exLink.MemoryShift + (Internal.x + Internal.RecordStart)*SIZEOF(Internal.RecordData), SIZEOF(Internal.RecordData));

				UIConnect.Output.StartTime[Internal.x] := Internal.RecordData.TimeStart;
				UIConnect.Output.EndTime[Internal.x] := Internal.RecordData.TimeEnd;
				UIConnect.Output.ShiftName[Internal.x] := Internal.RecordData.ShiftName;
				UIConnect.Output.CurrentUser[Internal.x] := Internal.RecordData.CurrentUser;
				UIConnect.Output.AdditionalData[Internal.x] := Internal.RecordData.AdditionalData;
				UIConnect.Output.TargetPieces[Internal.x] := Internal.RecordData.TargetPieces;
				UIConnect.Output.TotalPieces[Internal.x] := Internal.RecordData.TotalPieces;
				UIConnect.Output.GoodPieces[Internal.x] := Internal.RecordData.GoodPieces;
				UIConnect.Output.RejectPieces[Internal.x] := Internal.RecordData.RejectPieces;
				UIConnect.Output.BadPieceRate[Internal.x] := Internal.RecordData.BadPieceRate;
				UIConnect.Output.TotalTime[Internal.x] := Internal.RecordData.TotalTime;
				UIConnect.Output.ScheduledDowntime[Internal.x] := Internal.RecordData.ScheduledDowntime;
				UIConnect.Output.UnscheduledDowntime[Internal.x] := Internal.RecordData.UnscheduledDowntime;
				UIConnect.Output.Uptime[Internal.x] := Internal.RecordData.Uptime;
				UIConnect.Output.GoodProductionTime[Internal.x] := Internal.RecordData.GoodProductionTime;
				UIConnect.Output.NominalProductionTime[Internal.x] := Internal.RecordData.NominalProductionTime;
				UIConnect.Output.NominalProductionRate[Internal.x] := Internal.RecordData.NominalProductionTimeRate;
				UIConnect.Output.UnscheduledDowntimeRate[Internal.x] := Internal.RecordData.UnscheduledDowntimeRate;
				UIConnect.Output.ProductionRate[Internal.x] := Internal.RecordData.CurrentProductionRate;
				UIConnect.Output.JobName[Internal.x] := Internal.RecordData.JobName;

				Internal.x := Internal.x + 1;

				UNTIL (Internal.x = UI_SHIFT_LIST_IDX) OR (Internal.x + Internal.RecordStart >= Internal.RecordCount)
			END_REPEAT;

			exLink.RefreshShiftUI := FALSE;
			UIConnect.Output.PageUp := FALSE;
			UIConnect.Output.PageDown := FALSE;
			UIConnect.Output.StepUp := FALSE;
			UIConnect.Output.StepDown := FALSE;

			CreateLoggerEntry(exASSETINT_LOG_INFO, ADR('refresh shift done'), Logger);
			Internal.State := exASSETINT_STATE_IDLE;

			// -------------------------------------------------------------------------------------------
			// Error state
		exASSETINT_STATE_ERROR:
			IF EDGEPOS(ErrorReset) THEN
				Internal.StateError := exASSETINT_STATE_NONE;
				Internal.State := exASSETINT_STATE_INIT_1;
			END_IF
	END_CASE;
END_FUNCTION_BLOCK

// -------------------------------------------------------------------------------------------
// Shift timeline function block
FUNCTION_BLOCK exAssetIntTimelineUI
	// -------------------------------------------------------------------------------------------
	// Reset everything when enable is false
	IF NOT Enable THEN
		StatusID := ERR_FUB_ENABLE_FALSE;
		Active := FALSE;
		Internal.State := exASSETINT_STATE_INIT_1;
		CreateLoggerEntry(exASSETINT_LOG_INFO, ADR('function block disabled'), Logger);
		RETURN;
	END_IF

	CASE Internal.State OF

		// -------------------------------------------------------------------------------------------
		// Wait for enable
		exASSETINT_STATE_INIT_1:
			IF Enable THEN
				CreateLoggerEntry(exASSETINT_LOG_INFO, ADR('function block enabled'), Logger);

				// Check prerequisites, exLink and buffers
				IF NOT exAssetIntCheckPreq(exLink, Logger, ADR(Internal.State), ADR(StatusID), ADR(Info.Diag.StatusID)) THEN
					RETURN;
				END_IF

				// Reset error and status
				Error := FALSE;
				StatusID := ERR_OK;
				Internal.SortingStartTimeOld := UDINT_TO_DINT(16#FFFFFFFF);

				// Reset filter settings
				exAssetIntFilterReset(ADR(UIConnect.Filter));

				Internal.State := exASSETINT_STATE_IDLE;
			END_IF

			// -------------------------------------------------------------------------------------------
			// Wait for new event
		exASSETINT_STATE_IDLE:
			// Set status
			UIConnect.Status := exASSETINT_UI_STATUS_IDLE;
			Active := TRUE;

			// Handle dialog window
			Internal.State := exAssetIntFilterListUI(ADR(UIConnect.Filter), ADR(UIConnect.Status), Logger);

			// Handle sorting direction change
			IF UISetup.SortingStartTime <> Internal.SortingStartTimeOld AND exLink.RecordCount > 0 THEN
				Internal.State := exASSETINT_STATE_UI_BUFFER;
			END_IF
			Internal.SortingStartTimeOld := UISetup.SortingStartTime;

			// Handle page up and down
			exAssetIntScrollListUI(Internal.RecordCount, UI_TIMELINE_IDX, ADR(UIConnect.Output.PageUp), ADR(UIConnect.Output.PageDown), ADR(UIConnect.Output.StepUp), ADR(UIConnect.Output.StepDown), ADR(Internal.RecordStart), ADR(Internal.State));

			// Wait for core task to call update command
			IF exLink.RefreshTimelineUI AND exLink.RecordCount > 0 THEN
				Internal.State := exASSETINT_STATE_UI_BUFFER;
			END_IF

			// -------------------------------------------------------------------------------------------
			// Copy timeline data from global buffer to timeline buffer
		exASSETINT_STATE_UI_BUFFER:
			// Set status
			CreateLoggerEntry(exASSETINT_LOG_INFO, ADR('refresh timeline data'), Logger);
			UIConnect.Status := exASSETINT_UI_STATUS_UPDATE;

			// Generate timeline data
			Internal.RecordCount := exAssetIntBufferUI(exLink.MemoryTimeline, exLink, UISetup.SortingStartTime, UIConnect.Filter, RecordTypeTimeline);

			// Generate bar graph data
			Internal.TimeLongest := 0;
			FOR Internal.x := 0 TO Internal.RecordCount DO
				brsmemcpy(ADR(Internal.RecordData), exLink.MemoryTimeline + (Internal.x + Internal.RecordStart)*SIZEOF(Internal.RecordData), SIZEOF(Internal.RecordData));

				Internal.TimeSeconds := Internal.RecordData.TotalTime.Hours*60*60 + Internal.RecordData.TotalTime.Minutes*60 + Internal.RecordData.TotalTime.Seconds;

				IF Internal.TimeSeconds > Internal.TimeLongest THEN
					Internal.TimeLongest := Internal.TimeSeconds;
				END_IF
			END_FOR

			Internal.State := exASSETINT_STATE_UI_DATA;

			// -------------------------------------------------------------------------------------------
			// Transfer data from buffer to list array
		exASSETINT_STATE_UI_DATA:

			Internal.x := 0;
			brsmemset(ADR(UIConnect.Output), 0, SIZEOF(UIConnect.Output));
			IF Internal.RecordCount > 0 THEN
				REPEAT
					brsmemcpy(ADR(Internal.RecordData), exLink.MemoryTimeline + (Internal.x + Internal.RecordStart)*SIZEOF(Internal.RecordData), SIZEOF(Internal.RecordData));
					Internal.TimeSeconds := Internal.RecordData.TotalTime.Hours*60*60 + Internal.RecordData.TotalTime.Minutes*60 + Internal.RecordData.TotalTime.Seconds;

					UIConnect.Output.StartTime[Internal.x] := Internal.RecordData.TimeStart;
					UIConnect.Output.ShiftName[Internal.x] := Internal.RecordData.ShiftName;
					UIConnect.Output.JobName[Internal.x] := Internal.RecordData.JobName;
					UIConnect.Output.ProductionState[Internal.x] := UDINT_TO_UINT(Internal.RecordData.EventType) - 2;
					UIConnect.Output.Duration[Internal.x] := Internal.RecordData.TotalTime;
					UIConnect.Output.Reason[Internal.x] := Internal.RecordData.AdditionalData;
					UIConnect.Output.DurationBar[Internal.x].Duration := REAL_TO_UDINT(UDINT_TO_REAL(Internal.TimeSeconds)/UDINT_TO_REAL(Internal.TimeLongest)*100);

					IF Internal.RecordData.EventType = RecordTypeUptime THEN
						UIConnect.Output.DurationBar[Internal.x].Color := 2;
					ELSIF Internal.RecordData.EventType = RecordTypeDowntimeScheduled THEN
						UIConnect.Output.DurationBar[Internal.x].Color := 14;
					ELSIF Internal.RecordData.EventType = RecordTypeDowntimeUnscheduled THEN
						UIConnect.Output.DurationBar[Internal.x].Color := 51;
					END_IF

					Internal.x := Internal.x + 1;

					UNTIL (Internal.x = UI_TIMELINE_IDX) OR (Internal.x + Internal.RecordStart >= Internal.RecordCount)
				END_REPEAT;
			END_IF

			exLink.RefreshTimelineUI := FALSE;
			UIConnect.Output.PageUp := FALSE;
			UIConnect.Output.PageDown := FALSE;
			UIConnect.Output.StepUp := FALSE;
			UIConnect.Output.StepDown := FALSE;

			CreateLoggerEntry(exASSETINT_LOG_INFO, ADR('refresh timeline done'), Logger);
			Internal.State := exASSETINT_STATE_IDLE;

			// -------------------------------------------------------------------------------------------
			// Error state
		exASSETINT_STATE_ERROR:
			IF EDGEPOS(ErrorReset) THEN
				Internal.StateError := exASSETINT_STATE_NONE;
				Internal.State := exASSETINT_STATE_INIT_1;
			END_IF
	END_CASE;
END_FUNCTION_BLOCK

// -------------------------------------------------------------------------------------------
// Generate buffer data for job, shift or timeline
FUNCTION exAssetIntBufferUI
	brsmemset(Memory, 0, CORE_EVENT_NUM_MAX*SIZEOF(RecordData));
	IF exLink.RecordCount > 0 THEN
		REPEAT
			// Check sorting direction
			IF SortingStartTime = exASSETINT_SORTING_ASC THEN
				brsmemcpy(ADR(RecordData), exLink.MemoryDb + y*SIZEOF(RecordData), SIZEOF(RecordData));
			ELSE
				brsmemcpy(ADR(RecordData), exLink.MemoryDb + (exLink.RecordCount - y - 1)*SIZEOF(RecordData), SIZEOF(RecordData));
			END_IF

			// Data must match event type
			// or eventy type is shift and data is shift or job and flag is set to show job and shift data together
			// or eventy type is timeline and data timeline data (>= RecordTypeNoShift)
			IF (RecordData.EventType = EventType) OR
			   (EventType = RecordTypeShift AND UI_SHIFT_SHOW_JOBS AND (RecordData.EventType = RecordTypeShift OR RecordData.EventType = RecordTypeJob)) OR
     		   (EventType = RecordTypeTimeline AND RecordData.EventType >= RecordTypeNoShift) THEN
				// Only transfer data that matches filter
				IF (NOT Filter.Current.From.Enable AND NOT Filter.Current.Until.Enable) OR
					(Filter.Current.From.Enable AND Filter.Current.From.DateTime <= RecordData.TimeStart AND NOT Filter.Current.Until.Enable) OR
					(NOT Filter.Current.From.Enable AND Filter.Current.Until.Enable AND Filter.Current.Until.DateTime >= RecordData.TimeEnd) OR
					(Filter.Current.From.Enable AND Filter.Current.From.DateTime <= RecordData.TimeStart AND Filter.Current.Until.Enable AND Filter.Current.Until.DateTime >= RecordData.TimeEnd) THEN

					brsmemcpy(Memory + RecordCount*SIZEOF(RecordData), ADR(RecordData), SIZEOF(RecordData));
					RecordCount := RecordCount + 1;
				END_IF
			END_IF

			y := y + 1;

			UNTIL (y = exLink.RecordCount)
		END_REPEAT;
	END_IF

	exAssetIntBufferUI := RecordCount;
END_FUNCTION

// -------------------------------------------------------------------------------------------
// Check prerequisites, exLink and buffers
FUNCTION exAssetIntCheckPreq
	// Make sure we have remanent buffer
	IF ADR(exLink) = 0 THEN
		// Set status, remember state, go to error state
		StatusID := CreateErrorState(ERR_ASSET_LINK, ADR('ERR: exLink is 0'), Logger, exCOM_SEV_ERROR,  ADR(State), ADR(InfoDiagStatusID));
		exAssetIntCheckPreq := FALSE;
		RETURN;
	END_IF
	// Make sure we have temporary buffer
	IF exLink.MemoryDb = 0 OR exLink.MemoryJob = 0 OR exLink.MemoryTimeline = 0 THEN
		// Set status, remember state, go to error state
		StatusID := CreateErrorState(ERR_ASSET_TEMP_MEMORY, ADR('ERR: no temp memory'), Logger, exCOM_SEV_ERROR,  ADR(State), ADR(InfoDiagStatusID));
		exAssetIntCheckPreq := FALSE;
		RETURN;
	END_IF
	// Make sure core function block is active
	IF NOT exLink.IsCoreActive THEN
		// Set status, remember state, go to error state
		StatusID := CreateErrorState(exASSETINT_INF_WAIT_CORE_FB, ADR('ERR: core is not active'), Logger, exCOM_SEV_ERROR,  ADR(State), ADR(InfoDiagStatusID));
		exAssetIntCheckPreq := FALSE;
		RETURN;
	END_IF
	exAssetIntCheckPreq := TRUE;
END_FUNCTION

// -------------------------------------------------------------------------------------------
// Handle list scrolling
FUNCTION exAssetIntScrollListUI
	// -------------------------------------------------------------------------------------------
	// Handle page up and down
	IF PageUp THEN
		RecordStart := RecordStart - ListMaxCount;
		State := exASSETINT_STATE_UI_DATA;
	END_IF
	IF PageDown THEN
		RecordStart := RecordStart + ListMaxCount;
		State := exASSETINT_STATE_UI_DATA;
	END_IF

	// -------------------------------------------------------------------------------------------
	// Handle step up and down
	IF StepUp THEN
		RecordStart := RecordStart - 1;
		State := exASSETINT_STATE_UI_DATA;
	END_IF
	IF StepDown THEN
		RecordStart := RecordStart + 1;
		State := exASSETINT_STATE_UI_DATA;
	END_IF

	// -------------------------------------------------------------------------------------------
	// Correction for step/page up/down
	IF RecordStart + ListMaxCount > UDINT_TO_DINT(RecordCount) THEN
		RecordStart := RecordCount - ListMaxCount;
	END_IF
	IF RecordStart < 0 THEN
		RecordStart := 0;
	END_IF

	PageUp := FALSE;
	PageDown := FALSE;
	StepUp := FALSE;
	StepDown := FALSE;

	exAssetIntScrollListUI := TRUE;
END_FUNCTION

// -------------------------------------------------------------------------------------------
// Reset filter settings
FUNCTION exAssetIntFilterReset
	Filter.DefaultLayerStatus := 0;
	Filter.Dialog.LayerStatus := 1;
	Filter.Dialog.From.Year := 1970;
	Filter.Dialog.From.Month := 1;
	Filter.Dialog.From.Day := 1;
	Filter.Dialog.Until.Year := 1970;
	Filter.Dialog.Until.Month := 1;
	Filter.Dialog.Until.Day := 1;

	exAssetIntFilterReset := TRUE;
END_FUNCTION

// -------------------------------------------------------------------------------------------
// Handle dialog window
FUNCTION exAssetIntFilterListUI
	// Open dialog window
	IF Filter.ShowDialog THEN
		CreateLoggerEntry(exASSETINT_LOG_INFO, ADR('show dialog window'), Logger);

		Filter.Dialog.LayerStatus := 0;
		Filter.DefaultLayerStatus := 2;
		Filter.ShowDialog := FALSE;
	END_IF

	// Dialog is open
	IF Filter.Dialog.LayerStatus = 0 THEN
		Status := exASSETINT_UI_STATUS_FILTER;

		// Button cancel
		IF Filter.Dialog.Cancel THEN
			CreateLoggerEntry(exASSETINT_LOG_INFO, ADR('dialog canceled'), Logger);

			Filter.Dialog.LayerStatus := 1;
			Filter.DefaultLayerStatus := 0;
			Filter.Dialog.Cancel := 0;
		END_IF
		// Button ok
		IF Filter.Dialog.Confirm THEN
			CreateLoggerEntry(exASSETINT_LOG_INFO, ADR('dialog ok'), Logger);

			DT_TO_DTStructure_0.year := Filter.Dialog.From.Year;
			DT_TO_DTStructure_0.month := Filter.Dialog.From.Month;
			DT_TO_DTStructure_0.day := Filter.Dialog.From.Day;
			DT_TO_DTStructure_0.hour := Filter.Dialog.From.Hour;
			DT_TO_DTStructure_0.minute := Filter.Dialog.From.Minute;
			Filter.Current.From.DateTime := DTStructure_TO_DT(ADR(DT_TO_DTStructure_0));
			Filter.Current.From.Enable := Filter.Dialog.From.Enable;

			DT_TO_DTStructure_0.year := Filter.Dialog.Until.Year;
			DT_TO_DTStructure_0.month := Filter.Dialog.Until.Month;
			DT_TO_DTStructure_0.day := Filter.Dialog.Until.Day;
			DT_TO_DTStructure_0.hour := Filter.Dialog.Until.Hour;
			DT_TO_DTStructure_0.minute := Filter.Dialog.Until.Minute;
			Filter.Current.Until.DateTime := DTStructure_TO_DT(ADR(DT_TO_DTStructure_0));
			Filter.Current.Until.Enable := Filter.Dialog.Until.Enable;

			Filter.Dialog.LayerStatus := 1;
			Filter.DefaultLayerStatus := 0;
			Filter.Dialog.Confirm := 0;

			exAssetIntFilterListUI := exASSETINT_STATE_UI_BUFFER;
			RETURN;
		END_IF
	END_IF
	exAssetIntFilterListUI := exASSETINT_STATE_IDLE;

END_FUNCTION
```

#### CreateMemory.st
```iecst
// -------------------------------------------------------------------------------------------
// Create internal memory
// -------------------------------------------------------------------------------------------
FUNCTION_BLOCK CreateMemory
	// -------------------------------------------------------------------------------------------
	// Reset everything when enable is false
	IF NOT Enable THEN
		DatObjCreate_0.enable := FALSE;
		DatObjCreate_0();

		MemoryType := exASSETINT_MEM_DB;
		Status := ERR_FUB_ENABLE_FALSE;
		State := 0;
		RETURN;
	END_IF

	CASE State OF
		// -------------------------------------------------------------------------------------------
		// Wait for enable
		0:
			IF Enable THEN
				Cnt := 0;
				TmpStr1 := 'AsDb_0';
				Status := ERR_FUB_BUSY;
				CreateLoggerEntry(exASSETINT_LOG_INFO, ADR('creating internal memory'), Logger);
				State := 1;
			END_IF

			// -------------------------------------------------------------------------------------------
			// Generate new data module
		1:
			DatObjCreate_0.enable := TRUE;
			DatObjCreate_0.pName := ADR(TmpStr1);
			DatObjCreate_0.len := Size;
			DatObjCreate_0.MemType := doTEMP;
			DatObjCreate_0.Option := doNO_CS;
			DatObjCreate_0();

			// Data module created successful
			IF DatObjCreate_0.status = ERR_OK THEN
				// Created working memory
				IF MemoryType = exASSETINT_MEM_DB THEN
					// Generate log entry
					TmpStr2 := 'create db memory module ok > ';
					brsstrcat(ADR(TmpStr2), ADR(TmpStr1));
					CreateLoggerEntry(exASSETINT_LOG_ALL, ADR(TmpStr2), Logger);

					// Reset memory, set up next memory
					brsmemset(DatObjCreate_0.pDatObjMem, 0, Size);
					Cnt := 0;
					MemoryDb := DatObjCreate_0.pDatObjMem;
					MemoryType := exASSETINT_MEM_JOB;
					TmpStr1 := 'AsWr_0';
				ELSIF MemoryType = exASSETINT_MEM_JOB THEN
					// Generate log entry
					TmpStr2 := 'create job memory module ok > ';
					brsstrcat(ADR(TmpStr2), ADR(TmpStr1));
					CreateLoggerEntry(exASSETINT_LOG_ALL, ADR(TmpStr2), Logger);

					// Reset memory, set up next memory
					brsmemset(DatObjCreate_0.pDatObjMem, 0, Size);
					Cnt := 0;
					MemoryJob := DatObjCreate_0.pDatObjMem;
					MemoryType := exASSETINT_MEM_SHIFT;
					TmpStr1 := 'AsSh_0';
				ELSIF MemoryType = exASSETINT_MEM_SHIFT THEN
					// Generate log entry
					TmpStr2 := 'create shift memory module ok > ';
					brsstrcat(ADR(TmpStr2), ADR(TmpStr1));
					CreateLoggerEntry(exASSETINT_LOG_ALL, ADR(TmpStr2), Logger);

					// Reset memory, set up next memory
					brsmemset(DatObjCreate_0.pDatObjMem, 0, Size);
					Cnt := 0;
					MemoryShift := DatObjCreate_0.pDatObjMem;
					MemoryType := exASSETINT_MEM_TIMELINE;
					TmpStr1 := 'AsTl_0';
				ELSIF MemoryType = exASSETINT_MEM_TIMELINE THEN
					// Generate log entry
					TmpStr2 := 'create timeline memory module ok > ';
					brsstrcat(ADR(TmpStr2), ADR(TmpStr1));
					CreateLoggerEntry(exASSETINT_LOG_ALL, ADR(TmpStr2), Logger);

					// Reset memory, finish up
					brsmemset(DatObjCreate_0.pDatObjMem, 0, Size);
					MemoryTimeline := DatObjCreate_0.pDatObjMem;
					Status := ERR_OK;
					State := 0;
				END_IF

				DatObjCreate_0.enable := FALSE;
				DatObjCreate_0();

				// Data module already exists
			ELSIF DatObjCreate_0.status = doERR_DUPOBJECT  THEN
				// Generate log entry
				TmpStr2 := 'module already exists > ';
				brsstrcat(ADR(TmpStr2), ADR(TmpStr1));
				CreateLoggerEntry(exASSETINT_LOG_ALL, ADR(TmpStr2), Logger);

				// Increase module number, generate new module name
				Cnt := Cnt + 1;
				IF Cnt < 9 THEN
					brsmemset(ADR(TmpStr1) + brsstrlen(ADR(TmpStr1)) - 1, 0, 1);
				ELSE
					brsmemset(ADR(TmpStr1) + brsstrlen(ADR(TmpStr1)) - 2, 0, 2);
				END_IF
				brsitoa(Cnt, ADR(TmpStr2));
				brsstrcat(ADR(TmpStr1), ADR(TmpStr2));

				DatObjCreate_0.enable := FALSE;
				DatObjCreate_0();

				// Error
			ELSIF DatObjCreate_0.status <> ERR_FUB_BUSY THEN
				Status := DatObjCreate_0.status;
				State := 0;
			END_IF

	END_CASE;

END_FUNCTION_BLOCK
```

#### WriteEventData.st
```iecst
// -------------------------------------------------------------------------------------------
// File version 1000
// -------------------------------------------------------------------------------------------
// Write event data
// -------------------------------------------------------------------------------------------
FUNCTION_BLOCK WriteEventData
	// -------------------------------------------------------------------------------------------
	// Reset everything when enable is false
	IF NOT Enable THEN
		Status := ERR_FUB_ENABLE_FALSE;
		State := 0;
	END_IF

	CASE State OF
		// -------------------------------------------------------------------------------------------
		// Wait for enable
		0:
			IF EDGEPOS(Enable) THEN
				brsmemcpy(ADR(RecordDataIntern), RecordData, SIZEOF(RecordDataIntern));

				// Reset function blocks
				FileOpen_0.enable := FALSE;
				FileOpen_0();
				FileCreate_0.enable := FALSE;
				FileCreate_0();
				FileWrite_0.enable := FALSE;
				FileWrite_0();
				FileClose_0.enable := FALSE;
				FileClose_0();

				// Generate file name
				RecordDataIntern.FileName := CORE_FOLDER_NAME;
				brsstrcat(ADR(RecordDataIntern.FileName), ADR('/event#'));
				brsitoa(RecordIndex, ADR(TmpStr1));
				brsstrcat(ADR(RecordDataIntern.FileName), ADR(TmpStr1));

				Status := ERR_FUB_BUSY;
				TmpStr1 := 'creating new event type > ';
				brsitoa(RecordDataIntern.EventType, ADR(TmpStr2));
				brsstrcat(ADR(TmpStr1), ADR(TmpStr2));
				CreateLoggerEntry(exASSETINT_LOG_INFO, ADR(TmpStr1), Logger);
				State := 1;
			END_IF

			// -------------------------------------------------------------------------------------------
			// Open file
		1:
			FileOpen_0.enable := TRUE;
			FileOpen_0.pDevice := ADR(Device);
			FileOpen_0.pFile := ADR(RecordDataIntern.FileName);
			FileOpen_0.mode := fiREAD_WRITE;
			FileOpen_0();

			// File opened successful
			IF FileOpen_0.status = ERR_OK THEN
				// Generate log entry
				TmpStr1 := 'open event file ok > ';
				brsstrcat(ADR(TmpStr1), ADR(RecordDataIntern.FileName));
				CreateLoggerEntry(exASSETINT_LOG_ALL, ADR(TmpStr1), Logger);

				// Remember ident go to next step
				Ident := FileOpen_0.ident;
				State := 3;

				// Create event file when it does not exist
			ELSIF FileOpen_0.status = fiERR_FILE_NOT_FOUND  THEN
				State := 2;

				// Error
			ELSIF FileOpen_0.status <> ERR_FUB_BUSY THEN
				Status := FileOpen_0.status;
				State := 0;
			END_IF

			// -------------------------------------------------------------------------------------------
			// Create file
		2:
			FileCreate_0.enable := TRUE;
			FileCreate_0.pDevice := ADR(Device);
			FileCreate_0.pFile := ADR(RecordDataIntern.FileName);
			FileCreate_0();

			// File created successful
			IF FileCreate_0.status = ERR_OK THEN
				// Generate log entry
				TmpStr1 := 'create event file ok > ';
				brsstrcat(ADR(TmpStr1), ADR(RecordDataIntern.FileName));
				CreateLoggerEntry(exASSETINT_LOG_ALL, ADR(TmpStr1), Logger);

				// Remember ident go to next step
				Ident := FileCreate_0.ident;
				State := 3;

				// Error
			ELSIF FileCreate_0.status <> ERR_FUB_BUSY THEN
				Status := FileCreate_0.status;
				State := 0;
			END_IF

			// -------------------------------------------------------------------------------------------
			// Write data
		3:
			// Add file name to record
			RecordDataIntern.CRC := CalcCrc(ADR(RecordDataIntern), SIZEOF(RecordDataIntern));

			FileWrite_0.enable := TRUE;
			FileWrite_0.ident := Ident;
			FileWrite_0.pSrc := ADR(RecordDataIntern);
			FileWrite_0.len := SIZEOF(RecordDataIntern);
			FileWrite_0();

			// File created successful
			IF FileWrite_0.status = ERR_OK THEN
				// Generate log entry
				TmpStr1 := 'write event file ok > ';
				brsstrcat(ADR(TmpStr1), ADR(RecordDataIntern.FileName));
				CreateLoggerEntry(exASSETINT_LOG_ALL, ADR(TmpStr1), Logger);

				// Go to next step
				State := 4;

				// Error
			ELSIF FileWrite_0.status <> ERR_FUB_BUSY THEN
				Status := FileWrite_0.status;
				State := 0;
			END_IF

			// -------------------------------------------------------------------------------------------
			// Close file
		4:
			FileClose_0.enable := TRUE;
			FileClose_0.ident := Ident;
			FileClose_0();

			// File created successful
			IF FileClose_0.status = ERR_OK THEN
				// Generate log entry
				TmpStr1 := 'close event file ok > ';
				brsstrcat(ADR(TmpStr1), ADR(RecordDataIntern.FileName));
				CreateLoggerEntry(exASSETINT_LOG_ALL, ADR(TmpStr1), Logger);

				// Finish up
				brsmemcpy(RecordData, ADR(RecordDataIntern), SIZEOF(RecordDataIntern));
				Status := ERR_OK;
				State := 0;

				// Error
			ELSIF FileClose_0.status <> ERR_FUB_BUSY THEN
				Status := FileClose_0.status;
				State := 0;
			END_IF
	END_CASE;

END_FUNCTION_BLOCK
```

#### ReadEventData.st
```iecst
// -------------------------------------------------------------------------------------------
// Read event data
// -------------------------------------------------------------------------------------------
FUNCTION_BLOCK ReadEventData
	// -------------------------------------------------------------------------------------------
	// Reset everything when enable is false
	IF NOT Enable THEN
		Status := ERR_FUB_ENABLE_FALSE;
		State := 0;
	END_IF

	// Speed up read by executing function block twice
	FOR Override:=0 TO 1 DO
		CASE State OF
			// -------------------------------------------------------------------------------------------
			// Wait for enable
			0:
				IF EDGEPOS(Enable) THEN
					// Reset function blocks
					DirOpen_0.enable := FALSE;
					DirOpen_0();
					DirReadEx_0.enable := FALSE;
					DirReadEx_0();
					DirClose_0.enable := FALSE;
					DirClose_0();
					FileOpen_0.enable := FALSE;
					FileOpen_0();
					FileRead_0.enable := FALSE;
					FileRead_0();
					FileClose_0.enable := FALSE;
					FileClose_0();

					// Generate folder name
					DirCount := 0;
					TimeFirst := 0;
					DirName := 'events0';

					Status := ERR_FUB_BUSY;
					StatusRead := ERR_OK;
					RecordCount := 0;
					CreateLoggerEntry(exASSETINT_LOG_INFO, ADR('reading all events'), Logger);
					State := 1;
				END_IF

			// -------------------------------------------------------------------------------------------
			// Start reading folder
			1:
				DirOpen_0.enable := TRUE;
				DirOpen_0.pDevice := ADR(Device);
				DirOpen_0.pName := ADR(DirName);
				DirOpen_0();

				// File created successful
				IF DirOpen_0.status = ERR_OK THEN
					// Generate log entry
					TmpStr1 := 'open dir > ';
					brsstrcat(ADR(TmpStr1), ADR(DirName));
					CreateLoggerEntry(exASSETINT_LOG_ALL, ADR(TmpStr1), Logger);

					// Go to next step
					State := 2;

				// Error
				ELSIF DirOpen_0.status <> ERR_FUB_BUSY THEN
					Status := DirOpen_0.status;
					State := 0;
				END_IF

			// -------------------------------------------------------------------------------------------
			// Read next file name
			2:
				DirReadEx_0.enable := TRUE;
				DirReadEx_0.ident := DirOpen_0.ident;
				DirReadEx_0.pData := ADR(FileInfo_0);
				DirReadEx_0.data_len := SIZEOF(FileInfo_0);
				DirReadEx_0();

				// New file found
				IF DirReadEx_0.status = ERR_OK THEN
					IF brsstrcmp(ADR(FileInfo_0.Filename), ADR('.')) <> 0 AND brsstrcmp(ADR(FileInfo_0.Filename), ADR('..')) <> 0 THEN
						// Generate log entry
						TmpStr1 := 'found file > ';
						brsstrcat(ADR(TmpStr1), ADR(FileInfo_0.Filename));
						CreateLoggerEntry(exASSETINT_LOG_ALL, ADR(TmpStr1), Logger);

						State := 4;
					END_IF

				// No more entries
				ELSIF DirReadEx_0.status = fiERR_NO_MORE_ENTRIES THEN
					// Generate log entry
					TmpStr1 := 'read all events ok ';
					brsstrcat(ADR(TmpStr1), ADR(DirName));
					CreateLoggerEntry(exASSETINT_LOG_ALL, ADR(TmpStr1), Logger);

					State := 3;

				// Error
				ELSIF DirReadEx_0.status <> ERR_FUB_BUSY THEN
					Status := DirReadEx_0.status;
					State := 0;
				END_IF

			// -------------------------------------------------------------------------------------------
			// Finish reading folder
			3:
				DirClose_0.enable := TRUE;
				DirClose_0.ident := DirOpen_0.ident;
				DirClose_0();

				// Directory closed successful
				IF DirClose_0.status = ERR_OK THEN
					// Generate log entry
					TmpStr1 := 'close dir ok > ';
					brsstrcat(ADR(TmpStr1), ADR(DirName));
					CreateLoggerEntry(exASSETINT_LOG_ALL, ADR(TmpStr1), Logger);

					// Open next directory, finish when all folders are created
					DirCount := DirCount + 1;
					IF DirCount >= CORE_EVENT_NUM_MAX / CORE_EVENT_DIR_MAX THEN
						Status := ERR_OK;
						State := 0;

					// Generate next folder name
					ELSE
						DirName := 'events';
						brsitoa(DirCount, ADR(TmpStr2));
						brsstrcat(ADR(DirName), ADR(TmpStr2));
						State := 1;
					END_IF

				// Error
				ELSIF DirClose_0.status <> ERR_FUB_BUSY THEN
					Status := DirClose_0.status;
					State := 0;
				END_IF

			// -------------------------------------------------------------------------------------------
			// Open event file
			4:
				// Generate file name
				FileName := DirName;
				brsstrcat(ADR(FileName), ADR('/'));
				brsstrcat(ADR(FileName), ADR(FileInfo_0.Filename));

				// Open file
				FileOpen_0.enable := TRUE;
				FileOpen_0.pDevice := ADR(Device);
				FileOpen_0.pFile := ADR(FileName);
				FileOpen_0.mode := fiREAD_ONLY;
				FileOpen_0();

				// File opened successful
				IF FileOpen_0.status = ERR_OK THEN
					// Generate log entry
					TmpStr1 := 'open event file ok > ';
					brsstrcat(ADR(TmpStr1), ADR(FileName));
					CreateLoggerEntry(exASSETINT_LOG_ALL, ADR(TmpStr1), Logger);

					// Make sure data has correct size
					IF FileOpen_0.filelen <> SIZEOF(RecordData) THEN
						TmpStr1 := 'data in event file has wrong size > ';
						brsstrcat(ADR(TmpStr1), ADR(FileName));
						CreateLoggerEntry(exASSETINT_LOG_ERROR, ADR(TmpStr1), Logger);
						StatusRead := ERR_ASSET_READ_RECORD_SIZE;

						State := 6;
					ELSE
						State := 5;
					END_IF

					// Error
				ELSIF FileOpen_0.status <> ERR_FUB_BUSY THEN
					Status := FileOpen_0.status;
					State := 0;
				END_IF

			// -------------------------------------------------------------------------------------------
			// Read event data
			5:
				FileRead_0.enable := TRUE;
				FileRead_0.ident := FileOpen_0.ident;
				FileRead_0.pDest := ADR(RecordData);
				FileRead_0.len := FileOpen_0.filelen;
				FileRead_0();

				// File read successful
				IF FileRead_0.status = ERR_OK THEN
					// Generate log entry
					TmpStr1 := 'read event file ok > ';
					brsstrcat(ADR(TmpStr1), ADR(FileName));
					CreateLoggerEntry(exASSETINT_LOG_INFO, ADR(TmpStr1), Logger);

					// Check CRC
					CRC := CalcCrc(ADR(RecordData), SIZEOF(RecordData));
					IF CRC <> RecordData.CRC THEN
						// Generate log entry
						TmpStr1 := 'read event file CRC error > ';
						brsstrcat(ADR(TmpStr1), ADR(FileName));
						CreateLoggerEntry(exASSETINT_LOG_ERROR, ADR(TmpStr1), Logger);
						StatusRead := ERR_ASSET_READ_CRC;
					ELSE
						// Insert record
						InsertEventData(Memory, RecordCount, RecordData);
						RecordCount := RecordCount + 1;
					END_IF

					State := 6;

					// Error
				ELSIF FileRead_0.status <> ERR_FUB_BUSY THEN
					Status := FileRead_0.status;
					State := 6;
				END_IF

			// -------------------------------------------------------------------------------------------
			// Close file
			6:
				FileClose_0.enable := TRUE;
				FileClose_0.ident := FileOpen_0.ident;
				FileClose_0();

				// File closed successful
				IF FileClose_0.status = ERR_OK THEN
					// Generate log entry
					TmpStr1 := 'close event file ok > ';
					brsstrcat(ADR(TmpStr1), ADR(FileName));
					CreateLoggerEntry(exASSETINT_LOG_ALL, ADR(TmpStr1), Logger);

					// Auto delete corrupt file
					IF StatusRead = ERR_ASSET_READ_RECORD_SIZE OR StatusRead = ERR_ASSET_READ_CRC THEN
						State := 7;
					// Abort if there was a previous error, else proceed with next file
					ELSIF Status <> ERR_FUB_BUSY THEN
						State := 0;
					ELSE
						State := 2;
					END_IF

				// Error
				ELSIF FileClose_0.status <> ERR_FUB_BUSY THEN
					Status := FileClose_0.status;
					State := 0;
				END_IF

			// -------------------------------------------------------------------------------------------
			// Delete corrupt file
			7:
				FileDelete_0.enable := TRUE;
				FileDelete_0.pDevice := ADR(Device);
				FileDelete_0.pName := ADR(FileName);
				FileDelete_0();

				// File delete successful
				IF FileDelete_0.status = ERR_OK THEN
					// Generate log entry
					TmpStr1 := 'delete corrupt event file ok > ';
					brsstrcat(ADR(TmpStr1), ADR(FileName));
					CreateLoggerEntry(exASSETINT_LOG_ALL, ADR(TmpStr1), Logger);

					Status := StatusRead;
					State := 0;

				// Error
				ELSIF FileDelete_0.status <> ERR_FUB_BUSY THEN
					Status := FileDelete_0.status;
					State := 0;
				END_IF
		END_CASE;
	END_FOR;

END_FUNCTION_BLOCK

FUNCTION InsertEventData
	x := 0;
	y := 0;
	sort := 0;

	// Set up start values for iteration
	IF RecordCount <> 0 THEN
		y := RecordCount - 1;
	END_IF
	x := y;

	// Start itteration	search
	WHILE y > 1 DO
		// Check current entry
		RecordMemory ACCESS Memory + x*SIZEOF(RecordData);
		sort := DiffDT(RecordData.TimeEnd, RecordMemory.TimeEnd);

		// Solve new search range
		IF y MOD 2 = 0 THEN
			y := y / 2;
		ELSE
			y := y / 2 + 1;
		END_IF

		// New range is lower or higher than current
		IF sort <> 16#FFFFFFFF THEN
			x := x + y;
			IF x > UINT_TO_INT(RecordCount) THEN
				x := UINT_TO_INT(RecordCount);
			END_IF
		ELSE
			x := x - y;
			IF x < 1 THEN
				x := 1;
			END_IF
		END_IF
	END_WHILE;

	// New entry is this, next or previous
	RecordMemory ACCESS Memory + x*SIZEOF(RecordData);
	sort := DiffDT(RecordData.TimeEnd, RecordMemory.TimeEnd);

	IF sort > 0 AND x <> UINT_TO_INT(RecordCount) THEN
		x := x + 1;
	ELSIF x > 0 THEN
		RecordMemory ACCESS Memory + (x - 1)*SIZEOF(RecordData);
		sort := DiffDT(RecordData.TimeEnd, RecordMemory.TimeEnd);
		IF sort = 16#FFFFFFFF THEN
			x := x - 1;
		END_IF
	END_IF

	// Move all entrys backwards and fill in new entry
	brsmemmove(Memory + (x + 1)*SIZEOF(RecordData), Memory + x*SIZEOF(RecordData), (RecordCount - x)*SIZEOF(RecordData));
	brsmemcpy(Memory + x*SIZEOF(RecordData), ADR(RecordData), SIZEOF(RecordData));

	InsertEventData := TRUE;
END_FUNCTION
```
